# B&R Automation Studio project Lab2
Automation Studio 4.5.2.102

## Configuration SampleText

### Task classes (Cpu.sw)
```
Cyclic#4:
  DoorCtrl <- DoorCtrl.prg
  ncsdcctrl <- ncsdcctrl.prg
Cyclic#7:
  LED <- LED.prg
NcDataObjects: acp10etxen <- acp10etxen.dob
Binaries: TCData, iomap, Role, sysconf, arconfig, asfw, User, ashwd
Libraries: sys_lib, Runtime, asstring, X64Lib, Acp10man, Acp10par, NcGlobal, GateCtrl
```

### Hardware
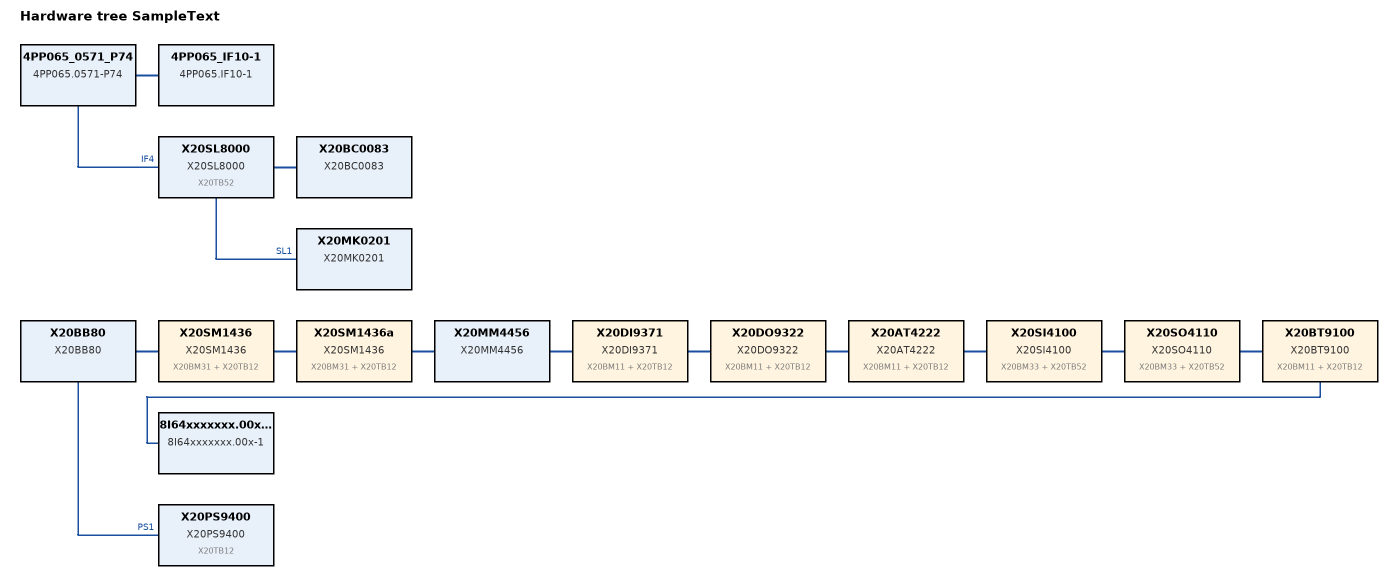
```
4PP065_0571_P74 : 4PP065.0571-P74 v1.1.2.0
  Connector IF4:
    EplInterfaceRedundant = 0
    EplEthInterfaceRedundant = 0
  Connector IF5:
    ActivateDevice = 1
    Mode = Manual
    InternetAddress = 10.0.1.10
    SubnetMask = 255.255.255.0
  ConfigurationID = labBR
  TimerDeviceType = EPLX2X
  TimerDevice = 4PP065_0571_P74.IF4
  TaskClassIdleTime = 2000
  Cyclic1Duration = 2000
  Cyclic1Tolerance = 0
  Cyclic1Output = 1
4PP065_IF10-1 : 4PP065.IF10-1 v1.0.3.0  [SS -> 4PP065_0571_P74.SS1]
8I64xxxxxxx.00x-1 : 8I64xxxxxxx.00x-1 v1.3.9.1  [X2X1 -> X20BT9100.X2X1 [Cable Type=X2XCable, Length=10, Version=1.0.0.2]]
  FunctionModel = Standard
  packedETAD = packed
  packedETI = packed
  packedCMDD = packed
  packedCMI = packed
X20AT4222 : X20AT4222 v1.2.3.0  [SS1 -> X20TB12e.SS; SL -> X20BM11c.SL1]
X20BB80 : X20BB80 v1.0.2.0
X20BC0083 : X20BC0083 v2.9.0.0  [PLK1 -> X20SL8000.PLK2 (NodeNumber=2) [Cable Type=PowerlinkCable, Length=10, Version=1.0.0.2]; SL -> X20BB80.SL1]
X20BM11 : X20BM11 v1.0.0.1  [X2X1 -> X20BM33a.X2X2]
X20BM11a : X20BM11 v1.0.0.1  [X2X1 -> X20MM4456.X2X2]
X20BM11b : X20BM11 v1.0.0.1  [X2X1 -> X20BM11a.X2X2]
X20BM11c : X20BM11 v1.0.0.1  [X2X1 -> X20BM11b.X2X2]
X20BM31 : X20BM31 v1.0.0.1  [X2X1 -> X20BB80.IF1]
X20BM31a : X20BM31 v1.0.0.1  [X2X1 -> X20BM31.X2X2]
X20BM33 : X20BM33 v1.0.0.4  [X2X1 -> X20BM11c.X2X2]
X20BM33a : X20BM33 v1.0.0.4  [X2X1 -> X20BM33.X2X2]
X20BT9100 : X20BT9100 v1.0.3.0  [SS1 -> X20TB12f.SS; SL -> X20BM11.SL1]
X20DI9371 : X20DI9371 v1.0.2.0  [SS1 -> X20TB12c.SS; SL -> X20BM11a.SL1]
X20DO9322 : X20DO9322 v1.0.3.0  [SS1 -> X20TB12d.SS; SL -> X20BM11b.SL1]
X20MK0201 : X20MK0201 v1.0.0.0  [SL -> X20SL8000.SL1]
X20MM4456 : X20MM4456 v1.1.5.0  [X2X1 -> X20BM31a.X2X2]
X20PS9400 : X20PS9400 v1.0.2.4  [SS1 -> X20TB12.SS; PS -> X20BB80.PS1]
X20SI4100 : X20SI4100 v1.10.1.1  [SS1 -> X20TB52.SS; SL -> X20BM33.SL1]
X20SL8000 : X20SL8000 v1.6.5.1  [PLK1 -> 4PP065_0571_P74.IF4 (NodeNumber=1) [Cable Type=PowerlinkCable, Length=10, Version=1.0.0.2]; PLK2 -> X20BC0083.PLK1 (NodeNumber=1) [Cable Type=PowerlinkCable, Length=10, Version=1.0.0.2]; SS1 -> X20TB52b.SS]
  SafeProject = SafeLOGIC-1
X20SM1436 : X20SM1436 v1.4.2.1  [SS1 -> X20TB12a.SS; SL -> X20BM31.SL1]
X20SM1436a : X20SM1436 v1.4.2.1  [SS1 -> X20TB12b.SS; SL -> X20BM31a.SL1]
X20SO4110 : X20SO4110 v1.10.1.1  [SS1 -> X20TB52a.SS; SL -> X20BM33a.SL1]
  SafeModuleID = 3
X20TB12 : X20TB12 v1.0.0.0
X20TB12a : X20TB12 v1.0.0.0
X20TB12b : X20TB12 v1.0.0.0
X20TB12c : X20TB12 v1.0.0.0
X20TB12d : X20TB12 v1.0.0.0
X20TB12e : X20TB12 v1.0.0.0
X20TB12f : X20TB12 v1.0.0.0
X20TB52 : X20TB52 v1.0.0.1
X20TB52a : X20TB52 v1.0.0.1
X20TB52b : X20TB52 v1.0.0.1
```

### IoMap.iom - 4PP065_0571_P74/IoMap.iom
```iecst
VAR_CONFIG
	::DoorCtrl:doorSM.sw1 AT %IX."X20DI9371".DigitalInput02;
	::DoorCtrl:doorSM.sw2 AT %IX."X20DI9371".DigitalInput03;
	::DoorCtrl:doorSM.sw3 AT %IX."X20DI9371".DigitalInput04;
	::DoorCtrl:doorSM.sw4 AT %IX."X20DI9371".DigitalInput05;
	::LED:Led1 AT %QX."X20DO9322".DigitalOutput02;
	::LED:Led2 AT %QX."X20DO9322".DigitalOutput03;
	::LED:Led3 AT %QX."X20DO9322".DigitalOutput04;
	::DoorCtrl:doorSM.direction AT %IX."X20DI9371".DigitalInput01;
	::DoorCtrl:ETAD AT %IW."8I64xxxxxxx.00x-1".ETAD_Input;
	::DoorCtrl:CMD AT %QW."8I64xxxxxxx.00x-1".CMDD_Output;
	::DoorCtrl:Speed AT %QW."8I64xxxxxxx.00x-1".LFRD_Output;
	::LED:Led4  AT %QX."X20DO9322".DigitalOutput05;
END_VAR
```

### Acp10cfg.ncc - 4PP065_0571_P74/Motion/Acp10cfg.ncc
```
NcConfiguration (Version=5.02.1, NcSwId=Acp10)
  ACP10CF1_typ:
    cnt_nettrc_rec_drive = 150
    bufsize_trace_upload = 1200
    tc_nc_man_task = Cyclic #1
    glob_pv_as_ncobject = Yes
    ncsys_dl_broadcast = Yes
    ncsys_dl_acp_reset = Yes
    safemc_log_err_to_ax = Yes
    network_init:
      ncsw_init_execute = Yes
      automatic_execute = No
      node_nr_warning = Yes
      net_err_before_ncact = Yes
    nettrc:
      enter_parsecrec = Yes
      enter_ncaction = Yes
      save_ring_startidx = No
    cam_prof_download:
      cam_dat_dl_parallel = No
      tc_cam_dl_parallel = Task class for NC Manager task
```

## Logical view

### Program Logical/DoorCtrl (ANSIC)

#### Main.cpp - Init, cyclic, exit code
```cpp
#include <bur/plctypes.h>

#ifdef _DEFAULT_INCLUDES
	#include <AsDefault.h>
#endif

// amount of memory to be allocated for heap storage must be specified for every ANSI C++ program with the bur_heap_size variable
unsigned long bur_heap_size = 0xFFFF;

void _INIT ProgramInit(void)
{
	// Insert code here

}

void _CYCLIC ProgramCyclic(void)
{
	FBGate(&doorSM);
	Speed = doorSM.Speed;
	doorSM.DriveCtrl.ETAD_Input = ETAD;
	CMD = doorSM.DriveCtrl.CMDD_Output;
	ledSM.state = doorSM.state;
	LedCtrl(&ledSM);
	L1 = ledSM.s1;
	L2 = ledSM.s2;
	L3 = ledSM.s3;
	L4 = ledSM.s4;
}

void _EXIT ProgramExit(void)
{
	// Insert code here

}
```

#### Variables.var - Local variables
```iecst
VAR
	doorSM : FBGate := (0);
	ledSM : LedCtrl := (0);
	ETAD : UINT := 0;
	Speed : INT := 0;
	CMD : UINT;
END_VAR
```

Listed in the project but not available here: Logical/DoorCtrl/Types.typ
